// TwinCAT 3 PLC project SupervisorPLC
// ProgramVersion: 3.1.4026.20
// libraries:
//   Tc2_ControllerToolbox, * (Beckhoff Automation GmbH)
//   Tc2_MC2, * (Beckhoff Automation GmbH)
//   Tc2_Standard, * (Beckhoff Automation GmbH)
//   Tc2_System, * (Beckhoff Automation GmbH)
//   Tc2_TcpIp, * (Beckhoff Automation GmbH)
//   Tc2_Utilities, * (Beckhoff Automation GmbH)
//   Tc3_EventLogger, * (Beckhoff Automation GmbH)
//   Tc3_JsonXml, * (Beckhoff Automation GmbH)
//   Tc3_Module, * (Beckhoff Automation GmbH)
// project tree:
//   Navitrol Supervisor/Common types/ ST_SectionHeader.TcDUT, ST_SupervisorHeader.TcDUT
//   Navitrol Supervisor/ FB_Supervisor.TcPOU
//   Navitrol Supervisor/Navitrol to Supervisor response/1100/ ST_1100_Position_initialization_started.TcDUT (not stored)
//   Navitrol Supervisor/Navitrol to Supervisor response/1101/Components/ E_1101_Initialization_result.TcDUT (not stored)
//   Navitrol Supervisor/Navitrol to Supervisor response/1101/ ST_1101_Position_initialized.TcDUT (not stored)
//   Navitrol Supervisor/Navitrol to Supervisor response/1116/ ST_1116_Motor_Control_Differential.TcDUT
//   Navitrol Supervisor/Navitrol to Supervisor response/1126/Components/ ST_1126_Omni_wheels_ref_struct.TcDUT (not stored), ST_1126_Supervisor_status_out.TcDUT (not stored)
//   Navitrol Supervisor/Navitrol to Supervisor response/1126/ ST_1126_Motor_control_omni_response.TcDUT (not stored)
//   Navitrol Supervisor/Navitrol to Supervisor response/3102/Components/ E_3102_Error_status.TcDUT, E_3102_Position_initialize_status.TcDUT, E_3102_State.TcDUT (not stored)
//   Navitrol Supervisor/Navitrol to Supervisor response/3102/Components/Sections/1/ ST_3102_1_General_section.TcDUT (not stored)
//   Navitrol Supervisor/Navitrol to Supervisor response/3102/ ST_3102_Navitrol_status.TcDUT
//   Navitrol Supervisor/Navitrol to Supervisor response/ Param_Supervisor_response.TcGVL, U_Recived_bytes_from_Navitrol.TcDUT
//   Navitrol Supervisor/Supervisor to Navitrol message/1001/ ST_1001_Initialize_position.TcDUT
//   Navitrol Supervisor/Supervisor to Navitrol message/1016/Components/ E_DriveControl.TcDUT (not stored)
//   Navitrol Supervisor/Supervisor to Navitrol message/1016/ ST_1016_Measurement_update_differential_drive.TcDUT (not stored)
//   Navitrol Supervisor/Supervisor to Navitrol message/1026/Components/ E_1026_Set_drive_mode.TcDUT (not stored), ST_1026_Omni_wheels_struct.TcDUT, ST_1026_Supervisor_status_bits.TcDUT
//   Navitrol Supervisor/Supervisor to Navitrol message/1026/ ST_1026_Measurement_update_generic_omni_drive.TcDUT (not stored)
//   Navitrol Supervisor/Supervisor to Navitrol message/3002/Components/ E_3002_Set_ESTOP.TcDUT, E_3002_Status.TcDUT (not stored)
//   Navitrol Supervisor/Supervisor to Navitrol message/3002/Components/Sections/2/Components/ E_3002_2_Enable_manual_control.TcDUT (not stored), E_3002_2_Inactive_Active.TcDUT
//   Navitrol Supervisor/Supervisor to Navitrol message/3002/Components/Sections/2/ ST_3002_2_Manual_section.TcDUT
//   Navitrol Supervisor/Supervisor to Navitrol message/3002/Components/Sections/6/Components/ E_3002_6_Joystick1_control_mode.TcDUT (not stored), E_3002_6_Joystick2_control_mode.TcDUT, E_3002_6_Steer_type_selection.TcDUT (not stored)
//   Navitrol Supervisor/Supervisor to Navitrol message/3002/Components/Sections/6/ ST_3002_6_Remote_control_section.TcDUT (not stored)
//   Navitrol Supervisor/Supervisor to Navitrol message/3002/Components/Sections/8/Components/ ST_3002_8_Binary_data.TcDUT (not stored), ST_3002_8_Error_status.TcDUT
//   Navitrol Supervisor/Supervisor to Navitrol message/3002/Components/Sections/8/ ST_3002_8_Battery_section.TcDUT (not stored)
//   Navitrol Supervisor/Supervisor to Navitrol message/3002/Components/Sections/ F_SetSectionHeaderInfo.TcPOU (not stored)
//   Navitrol Supervisor/Supervisor to Navitrol message/3002/ ST_3002_Supervisor_Status.TcDUT
//   Navitrol Supervisor/Supervisor to Navitrol message/ F_SetHeaderInfo.TcPOU
//   / PlcTask.TcTTO
//   POUs/ FB_StreamVelocity.TcPOU, MAIN.TcPOU
// real-time tasks:
//   TASK PlcTask: cycle T#1ms, priority 20, ADS port 350
// motion (NC):
//   TASK NC-Task 1 SAF: cycle T#2ms, priority 4, ADS port 501
//   TASK NC-Task 1 SVB: cycle T#10ms, priority 8, ADS port 511
//   AXIS LeftWheel (id 1)
//     General: UnitName=m
//     Dynamic: AccelerationMaximum=1, DecelerationMaximum=1, Acceleration=2222, Deceleration=2222, Jerk=224422000
//     Velo: SlowManual=0.6, FastManual=1, Maximum=2.2
//     OtherSettings: AllowMotionCmdToSlave=true
//     encoder EncType=1
//       EncPara: ScaleFactorNumerator=1e-07, EncMode=3
//     drive DrvType=5
//       Analog: VeloReferenz=2.2, TorqueSetpointScale=10, ScaleFactorActTorque=0.1
//       TimeComp: TaskDelayCycles=1
//     controller CtrType=1
//       CtrPara: PriorControlFactor=1
//         Observer: BandWidth=20
//   AXIS RightWheel (id 2)
//     General: UnitName=m
//     Dynamic: AccelerationMaximum=1, DecelerationMaximum=1, Acceleration=2222, Deceleration=2222, Jerk=224422000
//     Velo: SlowManual=0.6, FastManual=1, Maximum=2.2
//     OtherSettings: AllowMotionCmdToSlave=true
//     encoder EncType=1
//       EncPara: ScaleFactorNumerator=1e-07, EncMode=3
//     drive DrvType=5
//       Analog: VeloReferenz=2.2, TorqueSetpointScale=10, ScaleFactorActTorque=0.1
//       TimeComp: TaskDelayCycles=1
//     controller CtrType=1
//       CtrPara: PriorControlFactor=1
//         Observer: BandWidth=20
// variable links:
//   SupervisorPLC Instance <-> NC-Task 1 SAF/Axes/LeftWheel
//     PlcTask Inputs/MAIN.LeftWheel.NcToPlc <-> Outputs/ToPlc
//     PlcTask Outputs/MAIN.LeftWheel.PlcToNc <-> Inputs/FromPlc
//   SupervisorPLC Instance <-> NC-Task 1 SAF/Axes/RightWheel
//     PlcTask Inputs/MAIN.RightWheel.NcToPlc <-> Outputs/ToPlc
//     PlcTask Outputs/MAIN.RightWheel.PlcToNc <-> Inputs/FromPlc

CONFIGURATION SupervisorPLC
    RESOURCE PLC ON TwinCAT3
        TASK PlcTask(INTERVAL := T#1ms, PRIORITY := 20);
        PROGRAM MAIN WITH PlcTask : MAIN;
    END_RESOURCE
END_CONFIGURATION

// ---- Navitrol Supervisor/Common types/ST_SectionHeader.TcDUT
{attribute 'pack_mode' := '1'}
TYPE ST_SectionHeader :
	STRUCT
		Section_ID	   : UINT;
		Section_length : UDINT;
	END_STRUCT
END_TYPE

// ---- Navitrol Supervisor/Common types/ST_SupervisorHeader.TcDUT
{attribute 'pack_mode' := '1'}
//{attribute 'hide_all_locals'}
TYPE ST_SupervisorHeader :
	STRUCT
		Protocol_version : UINT;	
		Message_ID		 : UINT;
		Message_length	 : UDINT;
	END_STRUCT
END_TYPE
//When sending a message from Supervisor to Navitrol, this is populated using F_SetHeaderInfo.

// ---- Navitrol Supervisor/Navitrol to Supervisor response/1116/ST_1116_Motor_Control_Differential.TcDUT
{attribute 'pack_mode' := '1'}
TYPE ST_1116_Motor_Control_Differential EXTENDS ST_SupervisorHeader :
	STRUCT
		Message_number			: UDINT; //Identification number for individual messages. NOTE: This value must match with the latest Odometer update message number sent by the Supervisor.
		Speed_Left				: REAL;	 // Reference speed for left wheel (m/s)
		Speed_Right				: REAL;	 // 	Reference speed for right wheel (m/s)
		Errors_Stopping_driving : UINT;	 //0 no errors, 1 error stopping driving
	END_STRUCT
END_TYPE

// ---- Navitrol Supervisor/Navitrol to Supervisor response/3102/Components/E_3102_Error_status.TcDUT
{attribute 'qualified_only'}
{attribute 'strict'}
{attribute 'to_string'}
TYPE E_3102_Error_status :
(
	no_error := 0,
	error_on	:=1
)UINT;
END_TYPE

// ---- Navitrol Supervisor/Navitrol to Supervisor response/3102/Components/E_3102_Position_initialize_status.TcDUT
{attribute 'qualified_only'}
{attribute 'strict'}
{attribute 'to_string'}
TYPE E_3102_Position_initialize_status : (
		Failed	  := 0,
		Succeeded := 1
	) UINT;
END_TYPE

// ---- Navitrol Supervisor/Navitrol to Supervisor response/3102/ST_3102_Navitrol_status.TcDUT
{attribute 'pack_mode' := '1'}
TYPE ST_3102_Navitrol_status EXTENDS ST_SupervisorHeader :
	STRUCT
		DefaultSectionLength	   : UDINT;
		State					   : E_3102_State;
		X_coordinate			   : REAL; //In meters
		Y_coordinate			   : REAL; //In meters
		Heading					   : REAL; //Radians
		Level					   : DINT; //Level ID
		Speed					   : REAL; //m/s
		Position_initialize_status : E_3102_Position_initialize_status;
		Position_confidence		   : UINT; //Position confidence in percentage (1 - 100%)
		Error_status			   : E_3102_Error_status;
		//Additional sections can be added bellow - based on what is requested in the array of ST_3002_Supervisor_Status.Section_IDs 
		General_section			   : ST_3102_1_General_section;
	END_STRUCT
END_TYPE

// ---- Navitrol Supervisor/Navitrol to Supervisor response/U_Recived_bytes_from_Navitrol.TcDUT
// Bytes bucket to buffer received messages.
// Header info is parsed before being copied into the correct message structure.
// PLC logic is built expecting to receive the entire TCP message payload with one call to FB_SocketReceive.
// FB_SocketReceive will fragment the received data if the receive buffer is not large enough.
// Make sure this is large enough to fit the biggest received message.
TYPE U_Recived_bytes_from_Navitrol : UNION
		Header : ST_SupervisorHeader;
		Bytes  : ARRAY[0..Param_Supervisor_response.RecivedBytesBufferSize] OF UINT;
	END_UNION
END_TYPE

// ---- Navitrol Supervisor/Supervisor to Navitrol message/1001/ST_1001_Initialize_position.TcDUT
{attribute 'pack_mode' := '1'}
TYPE ST_1001_Initialize_position EXTENDS ST_SupervisorHeader:
	STRUCT
		X	   : REAL; //		X - map coordinate OF the AGV in meters
		Y	   : REAL; //		Y - map coordinate of the AGV in meters
		H	   : REAL; //		Heading of the AGV on the map in radians
		Level  : DINT; //	The level ID on which the AGV is located
	END_STRUCT
END_TYPE

// ---- Navitrol Supervisor/Supervisor to Navitrol message/1026/Components/ST_1026_Omni_wheels_struct.TcDUT
{attribute 'pack_mode' := '1'}
TYPE ST_1026_Omni_wheels_struct :
STRUCT
	Steer_angle	:REAL;
	Wheel_speed :REAL;
END_STRUCT
END_TYPE

// ---- Navitrol Supervisor/Supervisor to Navitrol message/1026/Components/ST_1026_Supervisor_status_bits.TcDUT
{attribute 'pack_mode' := '1'}
TYPE ST_1026_Supervisor_status_bits :
	STRUCT
		Error		   : BIT; //	When active ERROR_MOTOR_CONTROL_FAULT will be set.See error. in Glossary
		Emergency_stop : BIT; //	When active Navitrol will perform emergency stop and following two warnings will be triggered: WARNING_AGV_EM_STOP and WARNING_ESTOP_ACTIVE
		Soft_slow	   : BIT; //	When active Navitrol will perform soft slow.
		Soft_stop	   : BIT; //	When active Navitrol will perform soft stop.
		Reserved_4	   : BIT; //Not in use
		Reserved_5	   : BIT; //Not in use
		Reserved_6	   : BIT; //Not in use
		Brake_released : BIT; //	Informs Navitrol of the status of brakes.When not active hard stop will be enabled.
		Reserved_8_15  : BYTE; // Not in use
	END_STRUCT
END_TYPE

// ---- Navitrol Supervisor/Supervisor to Navitrol message/3002/Components/E_3002_Set_ESTOP.TcDUT
{attribute 'qualified_only'}
{attribute 'strict'}
{attribute 'to_string'}
TYPE E_3002_Set_ESTOP :
(
	Release_ESTOP := 0,
	Set_ESTOP:=1
)UINT;
END_TYPE

// ---- Navitrol Supervisor/Supervisor to Navitrol message/3002/Components/Sections/2/Components/E_3002_2_Inactive_Active.TcDUT
{attribute 'qualified_only'}
{attribute 'strict'}
{attribute 'to_string'}
TYPE E_3002_2_Inactive_Active : (
		Inactive := 0,
		Active	 := 1
	) UINT;
END_TYPE

// ---- Navitrol Supervisor/Supervisor to Navitrol message/3002/Components/Sections/2/ST_3002_2_Manual_section.TcDUT
{attribute 'pack_mode' := '1'}
TYPE ST_3002_2_Manual_section EXTENDS ST_SectionHeader :
	STRUCT
		Enable_manual_control : E_3002_2_Enable_manual_control;
		Forward				  : E_3002_2_Inactive_Active;
		Backward			  : E_3002_2_Inactive_Active;
		Left				  : E_3002_2_Inactive_Active;
		Right				  : E_3002_2_Inactive_Active;
		Drive_speed			  : REAL; //The manual drive speed reference in meters per second.
	END_STRUCT
END_TYPE

// ---- Navitrol Supervisor/Supervisor to Navitrol message/3002/Components/Sections/6/Components/E_3002_6_Joystick2_control_mode.TcDUT
{attribute 'qualified_only'}
{attribute 'strict'}
{attribute 'to_string'}
TYPE E_3002_6_Joystick2_control_mode : (
		No_control			:= 0,
		Enable_lift_control := 1
	)UINT;
END_TYPE

(*
Selects the joystick 2 control mode:
	0 - No control
Joystick 1 x and y values are ignored.
	1 - Enable lift control
	Navitrol activates manual mode.
*)

// ---- Navitrol Supervisor/Supervisor to Navitrol message/3002/Components/Sections/8/Components/ST_3002_8_Error_status.TcDUT
{attribute 'pack_mode' := '1'}
TYPE ST_3002_8_Error_status :
STRUCT
	Communication_error         : BIT; // BMS has lost the communication to the battery. *
	Configuration_error         : BIT; // Battery has not been correctly configured. *
	Undervoltage                : BIT; // Undervoltage detected. Operating voltage is low. Prepare to charge or replace the battery. *
	Overvoltage                 : BIT; // Overvoltage detected. Overvoltage is a sustained voltage that exceeds the normal steady state limits. *
	Overcurrent                 : BIT; // Overcurrent detected. Might be caused by overloading or short circuiting the battery. *
	Temperature_error           : BIT; // The temperature of the battery is at unsafe levels. * In addition, Navitrol will set ERROR_BATTERY_HIGH_TEMPERATURE
	Internal_defect             : BIT; // The battery has a defect and might not work properly. *
	Bad_state_of_health         : BIT; // The battery is worn down in use. It might not fully charge anymore. *
	Faulty_charger              : BIT; // The charger connected to the battery is not working. *
	Faulty_contactor            : BIT; // The contactor of the battery is not working. *
	Current_sensor_defect       : BIT; // The current sensor of the battery is not working. *
	Temperature_sensor_defect   : BIT; // The temperature sensor of the battery is not working. *
	Battery_cell_drift          : BIT; // Two or more battery cells are in imbalance. Can lead to over-charging or over-discharging harming the battery. *
	Charging_error              : BIT; // Error while charging the battery *
	Generic_error               : BIT; // This can be used to indicate that there is some other battery related error that is not listed above. *
	Reserved                    : BIT; // 0 - Not in use
END_STRUCT
END_TYPE

// ---- Navitrol Supervisor/Supervisor to Navitrol message/3002/ST_3002_Supervisor_Status.TcDUT
{attribute 'pack_mode' := '1'}
TYPE ST_3002_Supervisor_Status EXTENDS ST_SupervisorHeader :
	STRUCT
		Status			   : E_3002_Status			  := E_3002_Status.Ok;
		Set_Estop		   : E_3002_Set_ESTOP		  := E_3002_Set_ESTOP.Release_ESTOP;
		Number_of_sections : UINT					  := 1;	  //Number of sections requested in response message 3102. Change the size of Section_IDs's bellow to match.
		Section_IDs		   : ARRAY[1..1] OF UINT	  := [1]; //List of sections requested to send in the response message 3102. Make sure to add the expected recived message sections to the end of ST_3102_Navitrol_status
		Manual_section	   : ST_3002_2_Manual_section := (Enable_manual_control := E_3002_2_Enable_manual_control.Disable_control);
		Battery_section	   : ST_3002_8_Battery_section;
	END_STRUCT
END_TYPE

// ---- Navitrol Supervisor/Navitrol to Supervisor response/Param_Supervisor_response.TcGVL
{attribute 'qualified_only'}
VAR_GLOBAL CONSTANT
	RecivedBytesBufferSize	:UDINT:=5000;
END_VAR

// ---- POUs/MAIN.TcPOU
PROGRAM MAIN
VAR
	PowerLeftWheel		 : MC_Power;
	PowerRightWheel		 : MC_Power;
	LeftWheel			 : AXIS_REF;
	RightWheel			 : AXIS_REF;
	NavitrolInControl	 : BOOL := TRUE;
	StreamVeloLeftWheel	 : FB_StreamVelocity;
	StreamVeloRightWheel : FB_StreamVelocity;
	Supervisor			 : FB_Supervisor := (RemoteHost := '127.0.0.1', RemotePort := 2000);
END_VAR

Supervisor.st1016_Measurement_update_differential_drive.Odometry_left_wheel	 := TO_UDINT(LeftWheel.NcToPlc.ActPos * 10_000_000);
Supervisor.st1016_Measurement_update_differential_drive.Odometry_Right_wheel := TO_UDINT(RightWheel.NcToPlc.ActPos * 10_000_000);
Supervisor(Execute := TRUE);
PowerLeftWheel(Axis			   := LeftWheel,
			   Enable		   := TRUE,
			   Enable_Positive := TRUE,
			   Enable_Negative := TRUE,
			   Override		   := 100.0);

PowerRightWheel(Axis			:= RightWheel,
				Enable			:= TRUE,
				Enable_Positive := TRUE,
				Enable_Negative := TRUE,
				Override		:= 100.0);

StreamVeloLeftWheel(Axis		   := LeftWheel,
					Enable		   := NavitrolInControl,
					TargetVelocity := Supervisor.st1116_Motor_Control_Differential.Speed_Left);

StreamVeloRightWheel(Axis			:= RightWheel,
					 Enable			:= NavitrolInControl,
					 TargetVelocity := Supervisor.st1116_Motor_Control_Differential.Speed_Right);

END_PROGRAM

// ---- POUs/FB_StreamVelocity.TcPOU
FUNCTION_BLOCK FB_StreamVelocity
VAR_INPUT
	Axis			   : REFERENCE TO AXIS_REF;
	Enable			   : BOOL;
	TargetVelocity	   : LREAL; // Desired velocity setpoint (signed)
	Acceleration	   : LREAL := 0;
	Deceleration	   : LREAL := 0;
	Jerk			   : LREAL := 0;
	EnableSmoothing	   : BOOL  := TRUE;	   // Enable PT1 velocity smoothing
	FilterTimeConstant : TIME  := T#100MS; // PT1 time constant (tT1) - adjust for smoothing strength
END_VAR

VAR_OUTPUT
	Active			 : BOOL;
	Error			 : BOOL;
	ErrorID			 : UDINT;
	ActualVelocity	 : LREAL;
	Stopped			 : BOOL;
	WorkingVelocity  : LREAL;			  // The actual velocity setpoint being fed to NC (smoothed or raw)
	FilterError		 : BOOL;			  // PT1 filter error
	FilterErrorID	 : E_CTRL_ERRORCODES; // PT1 error code
END_VAR

VAR
	fbMoveVel1		   : MC_MoveVelocity;
	fbMoveVel2		   : MC_MoveVelocity;
	fbHalt			   : MC_Halt;
	bToggle			   : BOOL  := FALSE;
	rLastVelocity	   : LREAL := 0.0;
	bFirstCycle		   : BOOL  := TRUE;
	rVelocityTolerance : LREAL := 0.00001; // Threshold for issuing new command
	rAbsVelocity	   : LREAL;
	eDirection		   : MC_Direction;
	bStopActive		   : BOOL := FALSE;

	// PT1 smoothing
	fbPT1			 : FB_CTRL_PT1;
	stPT1Params		 : ST_CTRL_PT1_PARAMS;
	fbGetCycleTime	 : FB_CTRL_GET_TASK_CYCLETIME;
	bPT1Initialized	 : BOOL := FALSE;
END_VAR

// Initialize PT1 parameters once task cycle time is known
IF NOT bPT1Initialized THEN
	fbGetCycleTime(eMode := eCTRL_MODE_ACTIVE);
	IF fbGetCycleTime.bCycleTimeValid THEN
		stPT1Params.tTaskCycleTime := fbGetCycleTime.tTaskCycleTime;
		stPT1Params.tCtrlCycleTime := fbGetCycleTime.tTaskCycleTime; // Process every cycle
		bPT1Initialized			   := TRUE;
	ELSE
		// PT1 not ready yet - set defaults and exit early
		WorkingVelocity := TargetVelocity;
		FilterError		:= FALSE;
		FilterErrorID	:= eCTRL_ERROR_NOERROR;
		RETURN;
	END_IF
END_IF

// Update PT1 parameters from inputs (allows runtime tuning)
stPT1Params.fKp := 1;
stPT1Params.tT1 := FilterTimeConstant;

// Apply velocity smoothing if enabled
IF EnableSmoothing THEN
	fbPT1(fIn			:= TargetVelocity,
		  fManSyncValue := TargetVelocity,
		  bSync			:= FALSE,
		  eMode			:= eCTRL_MODE_ACTIVE,
		  bHold			:= FALSE,
		  stParams		:= stPT1Params);

	WorkingVelocity := fbPT1.fOut;
	FilterError		:= fbPT1.bError;
	FilterErrorID	:= fbPT1.eErrorId;
ELSE
	// No smoothing - sync PT1 to current value
	fbPT1(fIn			:= TargetVelocity,
		  fManSyncValue := TargetVelocity,
		  bSync			:= TRUE, // Sync to input when smoothing disabled
		  eMode			:= eCTRL_MODE_ACTIVE,
		  bHold			:= FALSE,
		  stParams		:= stPT1Params);

	WorkingVelocity := TargetVelocity;
	FilterError		:= fbPT1.bError;
	FilterErrorID	:= fbPT1.eErrorId;
END_IF

// Determine if we need to issue a new velocity command
IF Enable THEN
	// Check if we should stop (working velocity near zero)
	IF ABS(WorkingVelocity) < rVelocityTolerance THEN
		// Issue stop command if not already stopping
		IF NOT bStopActive THEN
			bStopActive	  := TRUE;
			rLastVelocity := 0.0;
		END_IF

		// Execute stop with aborting buffer mode
		fbHalt(Axis			:= Axis,
			   Execute		:= TRUE,
			   Deceleration := Deceleration,
			   Jerk			:= Jerk);

		// Reset velocity FBs
		fbMoveVel1(Axis := Axis, Execute := FALSE);
		fbMoveVel2(Axis := Axis, Execute := FALSE);
		Stopped := fbHalt.Done;
		Active	:= fbHalt.Busy;
		Error	:= fbHalt.Error;
		ErrorID := fbHalt.ErrorID;
	ELSE
		// We have a non-zero target velocity
		bStopActive := FALSE;

		// Reset stop FB
		fbHalt(Axis := Axis, Execute := FALSE);

		// Calculate absolute velocity and direction
		rAbsVelocity := ABS(WorkingVelocity);
		IF WorkingVelocity >= 0.0 THEN
			eDirection := MC_Positive_Direction;
		ELSE
			eDirection := MC_Negative_Direction;
		END_IF

		// Check if velocity setpoint has changed significantly
		IF ABS(WorkingVelocity - rLastVelocity) > rVelocityTolerance OR bFirstCycle THEN
			// Toggle between FB instances to achieve buffer aborting
			bToggle		  := NOT bToggle;
			rLastVelocity := WorkingVelocity;
			bFirstCycle	  := FALSE;
		END_IF

		// Execute alternating MoveVelocity commands with BufferMode := MC_Aborting
		fbMoveVel1(Axis			:= Axis,
				   Execute		:= Enable AND bToggle,
				   Velocity		:= rAbsVelocity,
				   Acceleration := Acceleration,
				   Deceleration := Deceleration,
				   Jerk			:= Jerk,
				   Direction	:= eDirection,
				   BufferMode	:= MC_Aborting);

		fbMoveVel2(Axis			:= Axis,
				   Execute		:= Enable AND NOT bToggle,
				   Velocity		:= rAbsVelocity,
				   Acceleration := Acceleration,
				   Deceleration := Deceleration,
				   Jerk			:= Jerk,
				   Direction	:= eDirection,
				   BufferMode	:= MC_Aborting);

		// Outputs
		Active	:= fbMoveVel1.Active OR fbMoveVel2.Active;
		Stopped := FALSE;
		Error	:= fbMoveVel1.Error OR fbMoveVel2.Error;
		ErrorID := SEL(fbMoveVel1.Error, fbMoveVel2.ErrorID, fbMoveVel1.ErrorID);
	END_IF

	ActualVelocity := Axis.NcToPlc.ActVelo;
ELSE
	// Reset when disabled
	fbMoveVel1(Axis := Axis, Execute := FALSE);
	fbMoveVel2(Axis := Axis, Execute := FALSE);
	fbHalt(Axis := Axis, Execute := FALSE);
	bFirstCycle := TRUE;
	bStopActive := FALSE;
	
	// Sync PT1 to zero when disabled
	fbPT1(fIn			:= 0.0,
		  fManSyncValue := 0.0,
		  bSync			:= TRUE,
		  eMode			:= eCTRL_MODE_ACTIVE,
		  bHold			:= FALSE,
		  stParams		:= stPT1Params);

	FilterError	  := fbPT1.bError;
	FilterErrorID := fbPT1.eErrorId;

	Active			:= FALSE;
	Stopped			:= FALSE;
	Error			:= FALSE;
	ErrorID			:= 0;
	WorkingVelocity := 0.0;
END_IF

END_FUNCTION_BLOCK

// ---- Navitrol Supervisor/FB_Supervisor.TcPOU
FUNCTION_BLOCK FB_Supervisor
VAR_INPUT
	RemoteHost									 : T_IPv4Addr := '127.0.0.1';
	RemotePort									 : UDINT	  := 2000;	  //Needs to match Navitrol parameter "supervisor_eth_port"
	CycleTime3002								 : TIME		  := T#500MS; //maximum interval 1 second
	CycleTime1026								 : TIME		  := T#10MS;  //This needs to match the Navitrol parameter "control_interval_us"
	Execute										 : BOOL;				  //Connect to Navitrol, and establish comuncations. If false, the socket is closed.
	st3002_Supervisor_Status					 : ST_3002_Supervisor_Status;
	st1016_Measurement_update_differential_drive : ST_1016_Measurement_update_differential_drive;

	//st1026_Measurement_update_generic_omni_drive : ST_1026_Measurement_update_generic_omni_drive;
	Initialize_position		   : BOOL; //Rising edge trigger to send a Initialize position command 
	st1001_Initialize_position : ST_1001_Initialize_position := (X := 21.23, Y := 36.95, H := 0, Level := 0);
END_VAR

VAR_OUTPUT
	st3102_Navitrol_status : ST_3102_Navitrol_status;

	//st1126_Motor_control_omni_response : ST_1126_Motor_control_omni_response;
	st1116_Motor_Control_Differential : ST_1116_Motor_Control_Differential;
	st1101_Position_initialized		  : ST_1101_Position_initialized;
	Busy							  : BOOL;
	Error							  : BOOL;
	ErrorID							  : UDINT;
END_VAR

VAR
	State : (INIT_FBs,
		CLOSE_OLD_SOCKETS,
		CONNECT_TO_Server,
		COMS_ACTIVE,
		CLOSE_CONNECTION);
	CloseAll : FB_SocketCloseAll;
	Connect	 : FB_SocketConnect;
	Close	 : FB_SocketClose;

	//Event logging
	FirstScan  : BOOL := TRUE;
	ErrorMsg   : FB_TcMessage;
	WarnMsg	   : FB_TcMessage;
	VerboseMsg : FB_TcMessage;
END_VAR

IF FirstScan THEN
	ErrorMsg.CreateEx(stEventEntry := TC_EVENTS.TcpIpComms.ErrorMsg, ipSourceInfo := 0);
	VerboseMsg.CreateEx(stEventEntry := TC_EVENTS.TcpIpComms.VerboseMsg, ipSourceInfo := 0);
	WarnMsg.CreateEx(stEventEntry := TC_EVENTS.TcpIpComms.WarnMsg, ipSourceInfo := 0);
	FirstScan := FALSE;
END_IF

CASE State OF
	INIT_FBs:
		CloseAll(bExecute := FALSE);
		Connect(bExecute := FALSE);
		Close(bExecute := FALSE);
		Busy := FALSE;
		IF Execute THEN
			Busy := TRUE;
			IF CycleTime3002 = T#0S OR CycleTime3002 > T#1S THEN
				ErrorMsg.ipArguments.Clear().AddString('Invalid input CycleTime3002');
				ErrorMsg.Send();
				Error := TRUE;
				RETURN;
			END_IF

			State := CLOSE_OLD_SOCKETS;
			Error := FALSE;
			VerboseMsg.ipArguments.Clear().AddString('Starting communications to:').AddString(RemoteHost).AddUDInt(RemotePort);
			VerboseMsg.Send();
		END_IF

	CLOSE_OLD_SOCKETS: //In the event of online change or download
		CloseAll(sSrvNetId := '', bExecute := TRUE, tTimeout := T#10S);
		IF NOT CloseAll.bBusy THEN
			CloseAll(bExecute := FALSE);
			State := CONNECT_TO_Server;
		END_IF

	CONNECT_TO_Server:
		Connect(sSrvNetId	:= '',
				sRemoteHost := RemoteHost,
				nRemotePort := RemotePort,
				bExecute	:= TRUE,
				tTimeout	:= T#4S);

		IF NOT Connect.bBusy THEN
			IF NOT Connect.bError THEN
				IF Connect.hSocket.handle <> 0 THEN
					State := COMS_ACTIVE;
					VerboseMsg.ipArguments.Clear().AddString('Connected to server:').AddString(RemoteHost).AddUDInt(RemotePort).AddString('Local port').AddUDInt(Connect.hSocket.localAddr.nPort);
					VerboseMsg.Send();
				END_IF
			ELSE
				Error := TRUE;
				State := INIT_FBs;
				ErrorMsg.ipArguments.Clear().AddString('Failed to connect to server:').AddString(RemoteHost).AddUDInt(RemotePort).AddString(', Error:').AddUDInt(Connect.nErrId);
				ErrorMsg.Send();
			END_IF

			Connect(bExecute := FALSE);
		END_IF

	COMS_ACTIVE:
		SendMsg3002();
		SengMeasurementUpdate();
		SendMsg1001();
		ReciveAllMsgsAndParse();
		IF NOT Execute THEN
			VerboseMsg.ipArguments.Clear().AddString('Connection closed by user');
			VerboseMsg.Send();
			State := CLOSE_CONNECTION;
		END_IF

	CLOSE_CONNECTION:
		Close(sSrvNetId := '',
			  hSocket	:= Connect.hSocket,
			  bExecute	:= TRUE,
			  tTimeout	:= T#4S);

		IF NOT Close.bBusy THEN
			Close(bExecute := FALSE);
			State := INIT_FBs;
		END_IF
END_CASE

METHOD INTERNAL ReciveAllMsgsAndParse : HRESULT
VAR_INST
	Receive								   : FB_SocketReceive;
	ReceiveBuffer						   : U_Recived_bytes_from_Navitrol;
	NumOf1100MsgRecived					   : UDINT;
	st1100_Position_initialization_started : ST_1100_Position_initialization_started;
	NumOf1101MsgRecived					   : UDINT;
	NumOf3102MsgRecived					   : UDINT;
	NumOf1116MsgRecived					   : UDINT;

	//NumOf1126MsgRecived					   : UDINT;
	UnknowMsgRecivedCounter : UDINT;
	UnknowMsg				: U_Recived_bytes_from_Navitrol;
END_VAR
Receive(sSrvNetId := '',
		hSocket	  := Connect.hSocket,
		cbLen	  := SIZEOF(ReceiveBuffer),
		pDest	  := ADR(ReceiveBuffer),
		bExecute  := TRUE,
		tTimeout  := T#10S);

IF NOT Receive.bBusy THEN
	IF Receive.nRecBytes <> 0 THEN
		IF Receive.nRecBytes = SIZEOF(ReceiveBuffer) THEN
			ErrorMsg.ipArguments.Clear().AddString('Recive buffer is not large enough! Please increase the size of "Param_Supervisor_response.RecivedBytesBufferSize');
			ErrorMsg.Send();
			State	:= CLOSE_CONNECTION;
			Error	:= TRUE;
			ErrorID := Global.TC_EVENTS.TcGeneralAdsEventClass.NoMemory.nEventId;
			RETURN;
		END_IF

		CASE ReceiveBuffer.Header.Message_ID OF //Check what message type is being recived - then copy it into the correct structure
			1100:
				NumOf1100MsgRecived := NumOf1100MsgRecived + 1;
				MEMCPY(destAddr := ADR(st1100_Position_initialization_started), srcAddr := ADR(ReceiveBuffer), n := SIZEOF(st1100_Position_initialization_started));
				VerboseMsg.ipArguments.Clear().AddString('Position initialization started');
				VerboseMsg.Send();

			1101:
				NumOf1101MsgRecived := NumOf1101MsgRecived + 1;
				MEMCPY(destAddr := ADR(st1101_Position_initialized), srcAddr := ADR(ReceiveBuffer), n := SIZEOF(st1101_Position_initialized));
				VerboseMsg.ipArguments.Clear().AddString('Position initialization finished');
				VerboseMsg.Send();

			1116:
				NumOf1116MsgRecived := NumOf1116MsgRecived + 1;
				MEMCPY(destAddr := ADR(st1116_Motor_Control_Differential), srcAddr := ADR(ReceiveBuffer), n := SIZEOF(st1116_Motor_Control_Differential));

				//1126:

				//	NumOf1126MsgRecived := NumOf1126MsgRecived + 1;

			//	MEMCPY(destAddr := ADR(st1126_Motor_control_omni_response), srcAddr := ADR(ReceiveBuffer), n := SIZEOF(st1126_Motor_control_omni_response));
			3102:
				NumOf3102MsgRecived := NumOf3102MsgRecived + 1;
				MEMCPY(destAddr := ADR(st3102_Navitrol_status), srcAddr := ADR(ReceiveBuffer), n := SIZEOF(st3102_Navitrol_status));

		ELSE
			UnknowMsgRecivedCounter := UnknowMsgRecivedCounter + 1;
			MEMCPY(destAddr := ADR(UnknowMsg), srcAddr := ADR(ReceiveBuffer), n := SIZEOF(UnknowMsg));
			WarnMsg.ipArguments.Clear().AddString('Unknow msg type recived with ID:').AddUInt(ReceiveBuffer.Header.Message_ID).AddString('Contents:').AddBlob(pData := ADR(ReceiveBuffer), cbData := TO_UINT(Receive.nRecBytes));
			WarnMsg.Send();
		END_CASE
	END_IF

	Receive(bExecute := FALSE);

	//Clear recive buffer
	MEMSET(destAddr := ADR(ReceiveBuffer), fillByte := 0, n := SIZEOF(ReceiveBuffer));
END_IF

IF Receive.bError THEN
	ErrorMsg.ipArguments.Clear().AddString('Failed to Receive, Error:').AddUDInt(Receive.nErrId);
	ErrorMsg.Send();
	State	:= CLOSE_CONNECTION;
	Error	:= TRUE;
	ErrorID := Receive.nErrId;
END_IF
END_METHOD

METHOD INTERNAL SendMsg1001 : HRESULT
VAR_INST
	rtInitialize_position : R_TRIG;
	Send1001			  : FB_SocketSend;
END_VAR
rtInitialize_position(CLK := Initialize_position);
IF rtInitialize_position.Q THEN
	F_SetHeaderInfo(st1001_Initialize_position);
	MEMSET(destAddr := ADR(st1101_Position_initialized), fillByte := 0, n := SIZEOF(st1101_Position_initialized)); //Clear old results
END_IF

Send1001(sSrvNetId := '',
		 hSocket   := Connect.hSocket,
		 cbLen	   := SIZEOF(st1001_Initialize_position),
		 pSrc	   := ADR(st1001_Initialize_position),
		 bExecute  := rtInitialize_position.Q,
		 tTimeout  := T#2S);

IF Send1001.bError THEN
	ErrorMsg.ipArguments.Clear().AddString('Failed to send 1001 Error:').AddUDInt(Send1001.nErrId);
	ErrorMsg.Send();
END_IF
END_METHOD

METHOD INTERNAL SendMsg3002 : HRESULT
VAR_INST
	Timer3002 : TON;
	Send3002  : FB_SocketSend;
END_VAR
Timer3002(IN := NOT Timer3002.Q, PT := CycleTime3002);
IF Timer3002.Q THEN
	F_SetHeaderInfo(st3002_Supervisor_Status);
	F_SetSectionHeaderInfo(st3002_Supervisor_Status.Manual_section);
	F_SetSectionHeaderInfo(st3002_Supervisor_Status.Battery_section);
	//Populate any added section headers here
END_IF

Send3002(sSrvNetId := '',
		 hSocket   := Connect.hSocket,
		 cbLen	   := SIZEOF(st3002_Supervisor_Status),
		 pSrc	   := ADR(st3002_Supervisor_Status),
		 bExecute  := Timer3002.Q,
		 tTimeout  := T#2S);

IF Send3002.bError THEN
	ErrorMsg.ipArguments.Clear().AddString('Failed to send 3002 Error:').AddUDInt(Send3002.nErrId);
	ErrorMsg.Send();
	State	:= CLOSE_CONNECTION;
	Error	:= TRUE;
	ErrorID := Send3002.nErrId;
END_IF
END_METHOD

METHOD INTERNAL SengMeasurementUpdate : HRESULT
VAR_INST
	Timer1026 : TON;
	Send1026  : FB_SocketSend;
END_VAR
Timer1026(IN := NOT Timer1026.Q, PT := CycleTime1026);
IF Timer1026.Q THEN
	//F_SetHeaderInfo(st1026_Measurement_update_generic_omni_drive);
	//st1026_Measurement_update_generic_omni_drive.Message_number := st1026_Measurement_update_generic_omni_drive.Message_number + 1;
	F_SetHeaderInfo(st1016_Measurement_update_differential_drive);
	st1016_Measurement_update_differential_drive.Message_number := st1016_Measurement_update_differential_drive.Message_number + 1;
	st1016_Measurement_update_differential_drive.Timestamp		:= st1016_Measurement_update_differential_drive.Timestamp + TO_UDINT(CycleTime1026);
END_IF

Send1026(sSrvNetId := '',
		 hSocket   := Connect.hSocket,
		 cbLen	   := SIZEOF(st1016_Measurement_update_differential_drive),
		 pSrc	   := ADR(st1016_Measurement_update_differential_drive),
		 //cbLen	   := SIZEOF(st1026_Measurement_update_generic_omni_drive),

		 //pSrc	   := ADR(st1026_Measurement_update_generic_omni_drive),
		 bExecute := Timer1026.Q,
		 tTimeout := T#2S);

IF Send1026.bError THEN
	ErrorMsg.ipArguments.Clear().AddString('Failed to send 1026 Error:').AddUDInt(Send1026.nErrId);
	ErrorMsg.Send();
	State	:= CLOSE_CONNECTION;
	Error	:= TRUE;
	ErrorID := Send1026.nErrId;
END_IF
END_METHOD

END_FUNCTION_BLOCK

// ---- Navitrol Supervisor/Supervisor to Navitrol message/F_SetHeaderInfo.TcPOU
//Use this to populate "ST_SupervisorHeader" in the message being sent from Supervisor to Navitrol
FUNCTION F_SetHeaderInfo : HRESULT;
VAR_INPUT
	Msg : ANY;
END_VAR

VAR
	MsgHeader			  : ST_SupervisorHeader;
	fbJsonDataType		  : FB_JsonReadWriteDataType;
	DataTypeName		  : STRING;
	Message_ID			  : UINT;
	GetDataTypeNameResult : HRESULT;
	i					  : INT;
	StartPos			  : INT;
	EndPos				  : INT;
	IDString			  : STRING;
	ParseSuccess		  : BOOL;
END_VAR

IF Msg.diSize < 0 THEN
	F_SetHeaderInfo := S_FALSE;
	RETURN;
END_IF

DataTypeName := fbJsonDataType.GetDataTypeNameByAddress(nData := TO_UDINT(Msg.diSize), pData := Msg.pValue, hrErrorCode => GetDataTypeNameResult);

// Parse Message_ID from DataTypeName (e.g., 'ST_3002_Supervisor_Status' -> 3002)
ParseSuccess := FALSE;
StartPos	 := FIND(DataTypeName, 'ST_');
IF StartPos > 0 THEN
	StartPos := StartPos + 3; // Move past 'ST_'

	// Find the next underscore after the ID
	EndPos := 0;
	FOR i := StartPos TO LEN(DataTypeName) DO
		IF MID(DataTypeName, 1, i) = '_' THEN
			EndPos := i;
			EXIT;
		END_IF
	END_FOR

	IF EndPos > StartPos THEN
		// Extract the ID substring
		IDString	 := MID(DataTypeName, EndPos - StartPos, StartPos);
		Message_ID	 := STRING_TO_UINT(IDString);
		ParseSuccess := TRUE;
	END_IF
END_IF

// Fallback if parsing fails
IF NOT ParseSuccess THEN
	Message_ID		:= 0;
	F_SetHeaderInfo := S_FALSE;
	RETURN;
END_IF

// All messages start with ST_SupervisorHeader
MsgHeader.Protocol_version := 4;
MsgHeader.Message_ID	   := Message_ID;
MsgHeader.Message_length   := TO_UDINT(Msg.diSize);

// Copy populated header into Msg
MEMCPY(destAddr := Msg.pValue, srcAddr := ADR(MsgHeader), n := SIZEOF(MsgHeader));
F_SetHeaderInfo := S_OK;

END_FUNCTION
